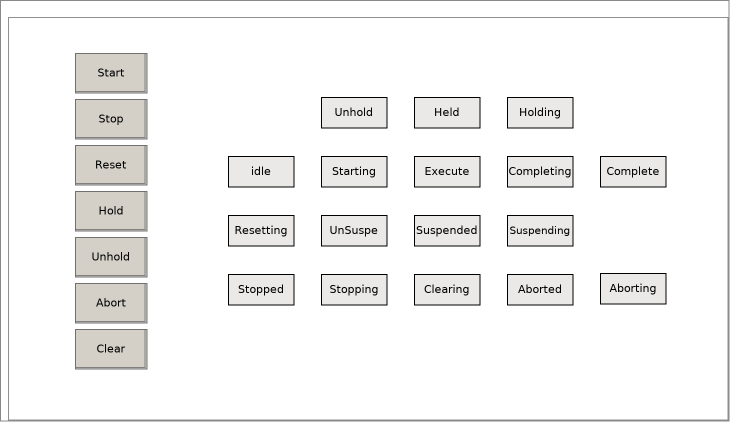
VISUALIZATION Vis_PackMlv3  // 730x422
VAR_IN_OUT
	PML3: PackMlv3_StateModel;
END_VAR
    GroupBox (8,9 720x411)
        RoundedRectangle (220,147 66x31), "idle", colour toggle: PML3.Sts_Idle
        Button (67,44 72x40), "Start"
            tap PML3.Cmd_Start
        Button (67,90 72x40), "Stop"
            tap PML3.Cmd_Stop
        Button (67,136 72x40), "Reset"
            tap PML3.Cmd_Reset
        Button (67,182 72x40), "Hold"
            tap PML3.Cmd_Hold
        Button (67,228 72x40), "Unhold"
            tap PML3.Cmd_UnHold
        Button (67,320 72x40), "Clear"
            tap PML3.Cmd_Clear
        Button (67,274 72x40), "Abort"
            tap PML3.Cmd_Abort
        RoundedRectangle (313,147 66x31), "Starting", colour toggle: PML3.Sts_Starting
        RoundedRectangle (406,147 66x31), "Execute", colour toggle: PML3.Sts_Execute
        RoundedRectangle (499,147 66x31), "Completing", colour toggle: PML3.Sts_Completing
        RoundedRectangle (592,147 66x31), "Complete", colour toggle: PML3.Sts_Complete
        RoundedRectangle (220,206 66x31), "Resetting", colour toggle: PML3.Sts_Resetting
        RoundedRectangle (313,88 66x31), "Unhold", colour toggle: PML3.Sts_UnHolding
        RoundedRectangle (220,265 66x31), "Stopped", colour toggle: PML3.Sts_Stopped
        RoundedRectangle (592,264 66x31), "Aborting", colour toggle: PML3.Sts_Aborting
    RoundedRectangle (321,215 66x31), "UnSuspe", colour toggle: PML3.Sts_UnSuspending
    RoundedRectangle (414,215 66x31), "Suspended", colour toggle: PML3.Sts_Suspended
    RoundedRectangle (507,215 66x31), "Suspending", colour toggle: PML3.Sts_Suspending
    RoundedRectangle (414,97 66x31), "Held", colour toggle: PML3.Sts_Held
    RoundedRectangle (507,97 66x31), "Holding", colour toggle: PML3.Sts_Holding
    RoundedRectangle (321,274 66x31), "Stopping", colour toggle: PML3.Sts_Stopping
    RoundedRectangle (414,274 66x31), "Clearing", colour toggle: PML3.Sts_Clearing
    RoundedRectangle (507,274 66x31), "Aborted", colour toggle: PML3.Sts_Aborted
END_VISUALIZATION

(* stored: Version 1.1.0.1, ProductVersion 3.1.4022.16
   Visu Vis_PackMlv3: Id {bef2400d-3ef2-4353-ab50-59856dfce416} *)
